// TIA Portal V18 export
DATA_BLOCK "VC_pulseHMI"   // DB344
{ S7_Optimized_Access := 'TRUE' }
VERSION : 0.1
// stored: AutoNumber true, DBAccessibleFromOPCUA true, IsOnlyStoredInLoadMemory false, IsRetainMemResEnabled false, IsWriteProtectedInAS false, MemoryReserve 100
   VAR
      "current Pulse VC1" : DInt;
      "current Pulse VC2" : DInt;
      "Previous Pulse VC1" : DInt;
      "Previous Pulse VC2" : DInt;
      "reset VC1" : Bool;
      "reset VC2" : Bool;
   END_VAR
BEGIN
END_DATA_BLOCK
